FUNCTION_BLOCK INTERNAL FB_InvocationControlTestTask EXTENDS FB_Task
VAR CONSTANT
    cDefaultCyclesToRun:        UDINT := 1;
END_VAR
VAR
    _nCyclesToRunIn:            UDINT;

    _nCyclesToRun:              UDINT := 10;
    _nCycleCounter:             UDINT;
END_VAR

PROPERTY nCycleCounter : UDINT
GET
nCycleCounter := THIS^._nCycleCounter;
END_GET
END_PROPERTY

METHOD PROTECTED OnStart
VAR_INPUT
END_VAR
IF THIS^._nCyclesToRunIn > 0 THEN
    THIS^._nCyclesToRun := THIS^._nCyclesToRunIn;
ELSE
    THIS^._nCyclesToRun := THIS^.cDefaultCyclesToRun;
END_IF
END_METHOD

METHOD Restore : I_Restorable
Restore := SUPER^.Restore();

THIS^._nCycleCounter := 0;
END_METHOD

METHOD Run
VAR_INPUT
END_VAR
IF THIS^.Execute() THEN
    THIS^._nCycleCounter := THIS^._nCycleCounter + 1;

    THIS^.DoneWhen(THIS^._nCycleCounter = THIS^._nCyclesToRun);
END_IF
END_METHOD

METHOD SetRunCondition : REFERENCE TO FB_InvocationControlTestTask
VAR_INPUT
    nCyclesToRun:        UDINT; // Number of cycles to run
END_VAR
SetRunCondition REF= THIS^;

THIS^._nCyclesToRunIn := nCyclesToRun;

THIS^.Invoke();
END_METHOD

END_FUNCTION_BLOCK

(* stored: Version 1.1.0.1, ProductVersion 3.1.4024.12
   POU FB_InvocationControlTestTask: Id {6d48c19b-0949-0447-175a-af01d4b69302}, SpecialFunc None
   Property nCycleCounter: Id {55855e17-67a2-06c2-1f3e-bf09c5bc6ad1}
   Get Get: Id {df7bef26-4887-0611-10a0-ae37acd4da44}
   Method OnStart: Id {35eb8f5c-047f-09ef-2ec4-647edcb9ddcf}
   Method Restore: Id {058b7504-7ac1-06de-1bfb-4add33843d09}
   Method Run: Id {f4236e24-17b7-009c-22d0-848f1ab39ee0}
   Method SetRunCondition: Id {8135ce41-7159-0be6-1fbb-fceacd1bb4a5} *)
